// TwinCAT 3 PLC project CarlPlc
// ProgramVersion: 3.1.4022.1
// libraries:
//   Tc2_ModbusRTU, * (Beckhoff Automation GmbH)
//   Tc2_Standard, * (Beckhoff Automation GmbH)
//   Tc2_System, * (Beckhoff Automation GmbH)
//   Tc2_Utilities, * (Beckhoff Automation GmbH)
//   Tc3_Module, * (Beckhoff Automation GmbH)
//   BASIC,3.3.3.0,OSCAT
// project tree:
//   Common/ DetectEvent.TcPOU (not stored), GVL_Common.TcGVL, TasterEventStates.TcDUT (not stored), TasterEventType.TcDUT (not stored), LinearCalibration.TcDUT (not stored)
//   FlowRateSensor/ GVL_FlowControl.TcGVL (not stored), PRG_UpdateFlowRateSensor.TcPOU (not stored)
//   GasAnalysis/ GVL_GasAnalysis.TcGVL (not stored), PRG_GasAnalysis.TcPOU
//   GasSupply/ GVL_GasSupply.TcGVL (not stored), PRG_UpdateGasSupply.TcPOU
//   MotorControl/ GVL_MotorControl.TcGVL (not stored), PRG_UpdateMotor.TcPOU (not stored)
//   pHOrpControl/ EN_ModbusReadTarget.TcDUT (not stored), GVL_PhOrpControl.TcGVL (not stored), PRG_ReadModbusSensorData.TcPOU (not stored), PRG_UpdatePhControl.TcPOU (not stored)
//   / PlcTask.TcTTO
//   MAIN/ MAIN.TcPOU
//   ReactorPressureControl/ GVL_ReactorPressureControl.TcGVL, PRG_UpdatePressureSensor.TcPOU
//   RoomTempRh/ GVL_TempRHSensor.TcGVL (not stored), PRG_UpdateRoomTempRh.TcPOU (not stored)
//   Systemidentifikation/ Messung1.TcPOU, Messung2.TcPOU
//   TemperatureControl/ EN_TempControlMode.TcDUT (not stored), GVL_TemperatureControl.TcGVL, FUN_ComputeMovingSetPoint.TcPOU (not stored), PRG_UpdateTemperatureControl.TcPOU
//   TemperatureControl/PID/ CLK_PRG.TcPOU (not stored), FB_PWM.TcPOU, FT_DERIV.TcPOU (not stored), FT_PIDWL.TcPOU (not stored), FT_PIWL.TcPOU (not stored), PWM_DC.TcPOU (not stored), TP_X.TcPOU, T_PLC_MS.TcPOU, T_PLC_US.TcPOU (not stored)
// real-time tasks:
//   TASK PlcTask: cycle T#10ms, priority 20, ADS port 350
// I/O:
//   DEVICE Device 1 (EtherCAT), AmsNetId 5.54.16.198.2.1
//     Term 1 (EK1200) [EK1200-5000 EtherCAT Power supply (2A E-Bus)]
//       Term 2 (EL3014) Motor Speed In [EL3014 4Ch. Ana. Input 0-20mA DIFF]
//       Term 3 (EL4004) Motor Speed Out [EL4004 4Ch. Ana. Output 0-10V, 12bit]
//       Term 4 (EL2004) DO Heating Cooling [EL2004 4Ch. Dig. Output 24V, 0.5A]
//       Term 5 (EL2004) DO Gassing Valves [EL2004 4Ch. Dig. Output 24V, 0.5A]
//       Term 6 (EL2004) DO Motor Control Out [EL2004 4Ch. Dig. Output 24V, 0.5A]
//       Term 7 (EL6021) PhModbus [EL6021 Interface (RS422/485)]
//       Term 8 (EL6021) OrpModbus [EL6021 Interface (RS422/485)]
//       Term 21 (EL1004) DI Gas Analysis [EL1004 4Ch. Dig. Input 24V, 3ms]
//       Term 18 (EL3052) AI Pressure Flow [EL3052 2Ch. Ana. Input 4-20mA]
//       Term 24 (EL3052) AI Heating Cooling [EL3052 2Ch. Ana. Input 4-20mA]
//       Term 10 (EL9184) [EL9184 Potential Connection, 8 x 24V, 8 x Ground]
//       Term 26 (EL3044) [EL3044 4Ch. Ana. Input 0-20mA]
//       Term 9 (EL9011) [EL9011 End Terminal]
// variable links:
//   CarlPlc/CarlPlc Instance <-> Device 1 (EtherCAT)/Term 1 (EK1200)/Term 18 (EL3052) AI Pressure Flow
//     PlcTask Inputs/GVL_FlowControl.flowRateRawCounts <-> FlowRateSensor/FlowRateRaw
//     PlcTask Inputs/GVL_ReactorPressureControl.pressureRawCounts <-> PressureSensor/PressureSensorRaw
//   CarlPlc/CarlPlc Instance <-> Device 1 (EtherCAT)/Term 1 (EK1200)/Term 2 (EL3014) Motor Speed In
//     PlcTask Inputs/GVL_MotorControl.motorActualSpeed <-> AI Motor RPM/Value
//     PlcTask Inputs/GVL_TempRHSensor.roomRhRaw <-> AI Room RH/Value
//     PlcTask Inputs/GVL_TempRHSensor.roomTempRaw <-> AI Room Temp/Value
//   CarlPlc/CarlPlc Instance <-> Device 1 (EtherCAT)/Term 1 (EK1200)/Term 21 (EL1004) DI Gas Analysis
//     PlcTask Inputs/GVL_GasAnalysis.ch4FlowSensor <-> Flow Sensor CH4/Input
//     PlcTask Inputs/GVL_GasAnalysis.o2FlowSensor <-> Flow Sensor O2/Input
//   CarlPlc/CarlPlc Instance <-> Device 1 (EtherCAT)/Term 1 (EK1200)/Term 24 (EL3052) AI Heating Cooling
//     PlcTask Inputs/GVL_TemperatureControl.jacketTempRaw <-> AI Jacket Temp/Value
//   CarlPlc/CarlPlc Instance <-> Device 1 (EtherCAT)/Term 1 (EK1200)/Term 26 (EL3044)
//     PlcTask Inputs/GVL_GasAnalysis.ch4SensorRaw <-> AI CH4/Value
//     PlcTask Inputs/GVL_GasAnalysis.o2SensorRaw <-> AI O2/Value
//     PlcTask Inputs/GVL_GasSupply.gasSupplyPressureRaw <-> AI Gas Supply Pressure/Value
//   CarlPlc/CarlPlc Instance <-> Device 1 (EtherCAT)/Term 1 (EK1200)/Term 3 (EL4004) Motor Speed Out
//     PlcTask Outputs/GVL_MotorControl.motorTargetSpeed <-> MotorTargetSpeed/MotorTargetSpeed
//     PlcTask Outputs/GVL_PhOrpControl.acidPumpSpeedCount <-> AcidPumpSpeedCount/acidPumpSpeedCount
//   CarlPlc/CarlPlc Instance <-> Device 1 (EtherCAT)/Term 1 (EK1200)/Term 4 (EL2004) DO Heating Cooling
//     PlcTask Outputs/GVL_TemperatureControl.coldValve <-> ColdValve/Output
//     PlcTask Outputs/GVL_TemperatureControl.hotValve <-> HotValve/Output
//     PlcTask Outputs/GVL_TemperatureControl.pumpOn <-> PumpOn/Output
//     PlcTask Outputs/GVL_TemperatureControl.steriValve <-> SteriValve/Output
//   CarlPlc/CarlPlc Instance <-> Device 1 (EtherCAT)/Term 1 (EK1200)/Term 5 (EL2004) DO Gassing Valves
//     PlcTask Outputs/GVL_GasSupply.gasSupplyValve <-> GasSupplyValve/Output
//     PlcTask Outputs/GVL_ReactorPressureControl.reactorPressureInletValve <-> reactorPressureInlet/ReactorPressureInlet
//     PlcTask Outputs/GVL_ReactorPressureControl.reactorPressureOutletValve <-> reactorPressureOutlet/Output
//   CarlPlc/CarlPlc Instance <-> Device 1 (EtherCAT)/Term 1 (EK1200)/Term 6 (EL2004) DO Motor Control Out
//     PlcTask Outputs/GVL_MotorControl.motorReset <-> motorReset/Output
//     PlcTask Outputs/GVL_MotorControl.motorStart <-> motorStart/Output
//   CarlPlc/CarlPlc Instance <-> Device 1 (EtherCAT)/Term 1 (EK1200)/Term 7 (EL6021) PhModbus
//     PlcTask Inputs/GVL_Common.PhModbus.InData/D[{0..21}] <-> COM TxPDO-Map Inputs/Data In {0..21}  (22 links)
//     PlcTask Inputs/GVL_Common.PhModbus.InData/Status <-> COM TxPDO-Map Inputs/Status
//     PlcTask Outputs/GVL_Common.PhModbus.OutData/Ctrl <-> COM RxPDO-Map Outputs/Ctrl
//     PlcTask Outputs/GVL_Common.PhModbus.OutData/D[{0..21}] <-> COM RxPDO-Map Outputs/Data Out {0..21}  (22 links)
//   CarlPlc/CarlPlc Instance <-> Device 1 (EtherCAT)/Term 1 (EK1200)/Term 8 (EL6021) OrpModbus
//     PlcTask Inputs/GVL_Common.OrpModbus.InData/D[{0..21}] <-> COM TxPDO-Map Inputs/Data In {0..21}  (22 links)
//     PlcTask Inputs/GVL_Common.OrpModbus.InData/Status <-> COM TxPDO-Map Inputs/Status
//     PlcTask Outputs/GVL_Common.OrpModbus.OutData/Ctrl <-> COM RxPDO-Map Outputs/Ctrl
//     PlcTask Outputs/GVL_Common.OrpModbus.OutData/D[{0..21}] <-> COM RxPDO-Map Outputs/Data Out {0..21}  (22 links)

CONFIGURATION CarlPlc
    RESOURCE PLC ON TwinCAT3
        TASK PlcTask(INTERVAL := T#10ms, PRIORITY := 20);
        PROGRAM MAIN WITH PlcTask : MAIN;
    END_RESOURCE
END_CONFIGURATION

// ---- Common/GVL_Common.TcGVL
VAR_GLOBAL
	
	loopCounter					: INT := 0;
	
		
	(* pH, ORP, and integrated thermometers *)
	PhModbus					: ModbusRtuMaster_KL6x22B;
	OrpModbus 					: ModbusRtuMaster_KL6x22B;
	PhValueArrayIn				: ARRAY [0..9]OF REAL;
	TPhValueArrayIn				: ARRAY [0..9]OF REAL;
	OrpValueArrayIn				: ARRAY [0..9] OF REAL;
	TOrpValueArrayIn			: ARRAY [0..9] OF REAL;
	
	
	
	
	
	
	
	
END_VAR

// ---- ReactorPressureControl/GVL_ReactorPressureControl.TcGVL
VAR_GLOBAL
	
	(* gas in-flow valve *)	
	reactorPressureInletValve AT %Q*	: BOOL := FALSE;
	
	(* gas out-flow bypass valve *)
	reactorPressureOutletValve		AT %Q* 	: BOOL := FALSE;

	(* pressure sensor *)
	pressureRawCounts	AT %I*	: INT := 0;
	pressureSensorCalibration	: LinearCalibration := (scaleFactor := 2.1626297577854671280276816608997E-4, offset := -1.0);
	pressureBar					: REAL := 0.0;
	pressureStart				: BOOL := FALSE;
	pressureStop				: BOOL := FALSE;

END_VAR

VAR_GLOBAL PERSISTENT
	pressureSetBar				: REAL;
	pressureRunning				: BOOL := FALSE;
END_VAR

// ---- TemperatureControl/GVL_TemperatureControl.TcGVL
VAR_GLOBAL

	tPhCurrent					: REAL := 0.0;
	tPhLastReadingValid			: BOOL := FALSE;
	tOrpCurrent					: REAL := 0.0;
	tOrpLastReadingValid		: BOOL := FALSE;


	(* temperature control *)
	pumpOn				AT %Q* 	: BOOL := FALSE;
	coldValve			AT %Q* 	: BOOL := FALSE;
	hotValve			AT %Q* 	: BOOL := FALSE;
	steriValve			AT %Q*	: BOOL := FALSE; 
	
	jacketTempRaw		AT %I*	: INT;
	jacketTempC					: REAL := 0.0;
	jacketTempK					: REAL := 0.0;
	
	
	tempControlStop				: BOOL := FALSE;
	tempControlStart			: BOOL := FALSE;
	hotValveButton				: BOOL := FALSE;
	coldValveButton				: BOOL := FALSE;
	
	pumpIsRunning				: BOOL := FALSE;
	tempControlRunning			: BOOL := FALSE;
	tempSafetyEnabled			: BOOL := FALSE;
	
	steriStart					: BOOL := FALSE;
	steriStop					: BOOL := FALSE;
	steriRunning				: BOOL := FALSE;

	
	currentMeanTemp				: REAL := 0;
	currentTempValid			: BOOL := FALSE;
	(* target temp -> see retains *) 
	
	tempIsBelowSteriTemp		: BOOL := TRUE;
	(* target steri temp --> see retains *)	

	
END_VAR

VAR_GLOBAL PERSISTENT
	targetControlTemp			: REAL;
	targetSteriTemp				: REAL;
	targetSteriTimeMinutes		: INT;
	remainingSteriTimeMinutes	: REAL;
	
	
	remainingSteriTimeInMs		: DINT; (* 30 min in ms *)
	
	countTempSpikes				: INT;
	countValveMaxTimeExceeded	: INT;

	pidResetCounter				: INT;
END_VAR

// ---- MAIN/MAIN.TcPOU
PROGRAM MAIN
VAR


END_VAR

loopCounter := loopCounter + 1;

PRG_ReadModbusSensorData();			//Temperatur von der Ph-Sonde

(* PRG_HandleUserInputs(); *)

PRG_UpdateMotor();					//Rührmotor

//PRG_UpdateTemperatureControl();		

PRG_UpdatePressureSensor();
PRG_UpdateFlowRateSensor();

Messung1();
//Messung2();

//PRG_UpdatePhControl();
//PRG_UpdateGasSupply();			//Erste Messung nicht nötig
//PRG_UpdateRoomTempRh();			//In Messungen implementiert
//PRG_GasAnalysis();				//Nicht notwendig

END_PROGRAM

// ---- ReactorPressureControl/PRG_UpdatePressureSensor.TcPOU
PROGRAM PRG_UpdatePressureSensor
VAR
	evtPressureControlStart		: DetectEvent;
	evtPressureControlStop		: DetectEvent;
	
END_VAR

(* convert the pressure signal *)
pressureBar := INT_TO_REAL(pressureRawCounts)*pressureSensorCalibration.scaleFactor + pressureSensorCalibration.offset;


(* button events *)
evtPressureControlStart(newSignalValue := pressureStart);
evtPressureControlStop(newSignalValue := pressureStop);

IF evtPressureControlStart.eventDetected = TASTEVT_PositiveEdge THEN
	pressureStart := FALSE;
	pressureRunning := TRUE;
END_IF

IF evtPressureControlStop.eventDetected = TASTEVT_PositiveEdge THEN
	pressureStop := FALSE;
	pressureRunning := FALSE;
END_IF


(* controller *)
IF pressureRunning THEN
	IF pressureBar > pressureSetBar + 0.01  THEN
		reactorPressureInletValve := FALSE;
	END_IF
	
	IF pressureBar < pressureSetBar - 0.01 THEN
		reactorPressureInletValve := TRUE;
	END_IF
ELSE
	reactorPressureInletValve := FALSE;
END_IF

END_PROGRAM

// ---- Systemidentifikation/Messung1.TcPOU
PROGRAM Messung1
VAR
	//PWM Settings
	pwmPeriodinSec			: TIME 	:= T#25S;
	pwmDutyCycle			: REAL 	:= 0.0;	
	pwmOutputValveControl 	: FB_PWM;
	status 					: INT 	:= 0; 			//Status 0 : Initial 
													//Status 1 : Heating to Startpoint
													//Status 2 : Heating while recording
													//Status 3 : Cooling while recording
													//STatus is set manuelly
													
END_VAR


(*Temperature should be increased to a value in a first step. 
This is to serve as a 0 point. In the second step, the duty cycle is increased and the step response is recorded.  
The container is then closed. The same duty cycle is used.
Finally, the water is cooled with a DutyCycle of ... .
*)

(* jacket temperature input *)
jacketTempC := INT_TO_REAL(jacketTempRaw)/32768.0*200.0 -50.0;
(* room temperature input *) //Is not in use in TemperaturControl
roomTemp := (INT_TO_REAL(roomTempRaw)/32767.0)*100.0 - 40.0;  (* Sensor Range: -40°C to + 60°C *)



// DutyCycle - To get a startingTemp.
CASE status OF
	
	//------Initial - Status 0----------//
	0:
	(* Setting Valves & Pump off  *)
	pumpOn := FALSE;
	coldValve := FALSE;
	hotValve := FALSE;
	steriValve := FALSE;
	
	//------HEATING - Status 1----------//
	1:
	//Starting pump
	pumpOn := TRUE;
	
	//DutyCyle for startpoint
	pwmDutyCycle:= 20 ;
	pwmOutputValveControl(pwmCycleTime:=pwmPeriodinSec, pwmDutyCycle:=pwmDutyCycle); //Gets the Output
	hotValve := pwmOutputValveControl.Q;
	
	
	//------HEATING - Status 2----------//
	2:	
	//DutyCycle for step response
	pwmDutyCycle:= 40 ;
	pwmOutputValveControl(pwmCycleTime:=pwmPeriodinSec, pwmDutyCycle:=pwmDutyCycle); //Gets the Output
	hotValve := pwmOutputValveControl.Q;
	
	//------COOLING - Status 3----------//
	3:
	//Turning off hotValve
	hotValve := FALSE;
	
	//DutyCycle for cooling
	pwmDutyCycle:= 40 ;
	pwmOutputValveControl(pwmCycleTime:=pwmPeriodinSec, pwmDutyCycle:=pwmDutyCycle); //Gets the Output
	coldValve := pwmOutputValveControl.Q;
END_CASE

END_PROGRAM

// ---- TemperatureControl/PID/FB_PWM.TcPOU
FUNCTION_BLOCK FB_PWM
VAR_INPUT
	pwmCycleTime 		: TIME := T#10S;
	pwmDutyCycle		: REAL := 0.5;
	reset				: BOOL := FALSE;
END_VAR
VAR_OUTPUT
	Q					: BOOL := FALSE;
END_VAR
VAR
	pwmTimeInMs			: INT	:= 0;
	pwmTimer		: TON;
	pwmLowTimer			: TON;
	dutyCycleInMs		: TIME;
	test				: INT;
	internalReset 		: BOOL := FALSE;
END_VAR

IF pwmDutyCycle < 0 THEN
	pwmDutyCycle := 0.0;
END_IF

IF reset OR internalReset THEN
	pwmTimer(IN:= FALSE);
	reset := FALSE;
	internalReset := FALSE;
ELSE
	pwmTimeInMs := TIME_TO_INT(pwmCycleTime);
	IF Q THEN
		(* high  --> running falling timer *)
		dutyCycleInMs := INT_TO_TIME(REAL_TO_INT(INT_TO_REAL(pwmTimeInMs)*pwmDutyCycle));
		pwmTimer(IN:=TRUE, PT:=dutyCycleInMs);
		IF pwmTimer.Q THEN
			internalReset := TRUE;
			Q := FALSE;
		END_IF		
	ELSE
		(* low --> running rising timer *)
		dutyCycleInMs := INT_TO_TIME(REAL_TO_INT(INT_TO_REAL(pwmTimeInMs)*(1.0-pwmDutyCycle)));
		pwmTimer(IN:=TRUE, PT:=dutyCycleInMs);
		IF pwmTimer.Q THEN
			internalReset := TRUE;
			Q := TRUE;
		END_IF		
	END_IF
END_IF

END_FUNCTION_BLOCK

// ---- GasAnalysis/PRG_GasAnalysis.TcPOU
PROGRAM PRG_GasAnalysis
VAR
	evtGasAnalysisStartStop		: DetectEvent;
	evtGasAnalysisManualValve 	: DetectEvent;
END_VAR

ch4ValuemA := ch4SensorRaw*ch4CalibrationToMa.scaleFactor + ch4CalibrationToMa.offset;
ch4ValuePercent := (ch4ValuemA-4.0)*(100.0/16.0);

o2ValuemA := o2SensorRaw*o2CalibrationToMa.scaleFactor + o2CalibrationToMa.offset;
o2ValuePercent := (o2ValuemA-4.0)*(25.0/16.0);



(* CH4 Sensor Status*)
IF ch4ValuemA > 3.9 THEN
	(* running *)
	ch4SensorStatus := 4;
ELSIF (ch4ValuemA < 3.2 AND ch4ValuemA > 2.8) THEN
	(* startup *)
	ch4SensorStatus := 3;
ELSIF (ch4ValuemA < 2.2 AND ch4ValuemA > 1.8) THEN
	(* beam block *)
	ch4SensorStatus := 2;
ELSIF (ch4ValuemA < 1.2 AND ch4ValuemA > 0.8) THEN
	(* fault *)
	ch4SensorStatus := 1;
ELSE
	(* offline *)
	ch4SensorStatus := 0;
END_IF

(* control switches *) 
evtGasAnalysisStartStop(newSignalValue := gasAnalysisControlStartStop);
IF evtGasAnalysisStartStop.eventDetected = TASTEVT_PositiveEdge THEN
	gasAnalysisControlRunning := TRUE;
END_IF

IF evtGasAnalysisStartStop.eventDetected = TASTEVT_NegativeEdge THEN
	gasAnalysisControlRunning := FALSE;
END_IF


IF gasAnalysisControlRunning THEN
	IF ch4ValuePercent > ch4ValuePercentSet  THEN
		gasAnalysisValveAutomatic := TRUE;
	END_IF
	
	IF ch4ValuePercent < ch4ValuePercentSet -1  THEN
		gasAnalysisValveAutomatic := FALSE;
	END_IF
ELSE 
	gasAnalysisValveAutomatic := FALSE;
END_IF


evtGasAnalysisManualValve(newSignalValue := gasAnalysisControlManual);
IF evtGasAnalysisManualValve.eventDetected = TASTEVT_PositiveEdge THEN
	gasAnalysisValveManual := TRUE;
END_IF

IF evtGasAnalysisManualValve.eventDetected = TASTEVT_NegativeEdge THEN
	gasAnalysisValveManual := FALSE;
END_IF

reactorPressureOutletValve := gasAnalysisValveManual OR gasAnalysisValveAutomatic;

END_PROGRAM

// ---- GasSupply/PRG_UpdateGasSupply.TcPOU
PROGRAM PRG_UpdateGasSupply
VAR
	evtGasSupplyStart		: DetectEvent;
	evtGasSupplyStop		: DetectEvent;
END_VAR

gasSupplyPressureBar := INT_TO_REAL(gasSupplyPressureRaw)*gasSupplyPressureSensorCalibration.scaleFactor + gasSupplyPressureSensorCalibration.offset;


(* button events *)
evtGasSupplyStart(newSignalValue := gasSupplyStart);
evtGasSupplyStop(newSignalValue := gasSupplyStop);

IF evtGasSupplyStart.eventDetected = TASTEVT_PositiveEdge THEN
	gasSupplyStart := FALSE;
	gasSupplyRunning := TRUE;
END_IF

IF evtGasSupplyStop.eventDetected = TASTEVT_PositiveEdge THEN
	gasSupplyStop := FALSE;
	gasSupplyRunning := FALSE;
END_IF


IF gasSupplyRunning THEN
	IF gasSupplyPressureBar > gasSupplyPressureSetBar + 0.1 THEN
		gasSupplyValve := FALSE;
	END_IF
	
	IF gasSupplyPressureBar < gasSupplyPressureSetBar - 0.1 THEN
		gasSupplyValve := TRUE;
	END_IF
 
END_IF

END_PROGRAM

// ---- Systemidentifikation/Messung2.TcPOU
PROGRAM Messung2
VAR
	//PWM Settings
	pwmPeriodinSec			: TIME 	:= T#25S;
	pwmDutyCycle			: REAL 	:= 0.0;	
	pwmOutputValveControl 	: FB_PWM;
	status 					: INT 	:= 0; 			//Status 0 : Initial 
													//Status 1 : Heating to Startpoint
													//Status 2 : Heating while recording
													//Status 3 : Cooling while recording
													//STatus is set manuelly
													
END_VAR


(*Temperature should be increased to a value in a first step. 
This is to serve as a 0 point. should be around 70°C
In the second step, the duty cycle is increased and the step response is recorded while the container is closed.
Finally, the water is cooled with a DutyCycle of ... .
*)

(* jacket temperature input *)
jacketTempC := INT_TO_REAL(jacketTempRaw)/32768.0*200.0 -50.0;
(* room temperature input *) //Is not in use in TemperaturControl
roomTemp := (INT_TO_REAL(roomTempRaw)/32767.0)*100.0 - 40.0;  (* Sensor Range: -40°C to + 60°C *)


// DutyCycle - To get a startingTemp.
CASE status OF
	
	//------Initial - Status 0----------//
	0:
	(* Setting Valves & Pump off  *)
	pumpOn := FALSE;
	coldValve := FALSE;
	hotValve := FALSE;
	steriValve := FALSE;
	
	//------HEATING - Status 1----------//
	1:
	//Starting pump
	pumpOn := TRUE;
	
	//DutyCyle for startpoint
	pwmDutyCycle:= 40 ;
	pwmOutputValveControl(pwmCycleTime:=pwmPeriodinSec, pwmDutyCycle:=pwmDutyCycle); //Gets the Output
	hotValve := pwmOutputValveControl.Q;
	
	
	//------HEATING - Status 2----------//
	2:	
	//Turning off the pump
	pumpOn := FALSE;
	
	//DutyCycle for step response
	pwmDutyCycle:= 80 ;
	pwmOutputValveControl(pwmCycleTime:=pwmPeriodinSec, pwmDutyCycle:=pwmDutyCycle); //Gets the Output
	steriValve := pwmOutputValveControl.Q;
	
	//------COOLING - Status 3----------//
	3:
	//Turning off hotValve & steriValve
	hotValve := FALSE;
	steriValve := FALSE;
	
	//DutyCycle for cooling
	pwmDutyCycle:= 40 ;
	pwmOutputValveControl(pwmCycleTime:=pwmPeriodinSec, pwmDutyCycle:=pwmDutyCycle); //Gets the Output
	coldValve := pwmOutputValveControl.Q;
END_CASE

END_PROGRAM

// ---- TemperatureControl/PID/TP_X.TcPOU
FUNCTION_BLOCK TP_X
VAR_INPUT
	IN : BOOL;
	PT : TIME;
END_VAR
VAR_OUTPUT
	Q : BOOL;
	ET : TIME;
END_VAR
VAR
	edge : BOOL;
	start : TIME;
	tx: TIME;
END_VAR

(*retriggerable edge triggered pulse similar to TP but with a retrigger function
if the pt input is 0 then output is always low.
*)

(* read system_time *)
tx := DWORD_TO_TIME(T_PLC_MS());

(* rising edge trigger *)
IF IN AND NOT edge THEN
	start := tx;
	Q := PT > t#0ms;
ELSIF Q THEN
	ET := tx - start;
	IF ET >= PT THEN
		Q := FALSE;
		ET := t#0ms;
	END_IF;
END_IF;
edge := IN;

END_FUNCTION_BLOCK

// ---- TemperatureControl/PID/T_PLC_MS.TcPOU
FUNCTION T_PLC_MS : DWORD
VAR CONSTANT
	debug : BOOL := 0;
	N : INT := 0;
	offset : DWORD := 0;
END_VAR
VAR
	tx : TIME;
END_VAR

(*T_PLC_MS reads the internal PLC timer and return the time, it has the advantage to be able to set a debug mode 
and speed up the counter to test the plc timer overrun which occurs every 50 days respectively 25 days at siemens S7
this routine also allows to correct the behavior of s7 where the internal plc counter will not count all 32 bits.

*)

tx := TIME();
T_PLC_MS := TIME_TO_DWORD(Tx);

IF debug THEN
	T_PLC_MS := (SHL(T_PLC_MS,N) OR SHL(DWORD#1,N)-1) + OFFSET;
END_IF;

END_FUNCTION

// ---- TemperatureControl/PRG_UpdateTemperatureControl.TcPOU
PROGRAM PRG_UpdateTemperatureControl
VAR
	tempControlMode				: EN_TempControlMode := EN_TempControlMode.TEMP_MODE_MANUAL;  

	(* Controller settings *)
	pwmPeriodinSec			: TIME := T#25S;
	pwmDutyCycle			: REAL := 0.0;	
	pwmOutputValveControl 	: FB_PWM;
	
	pidController			: FT_PIDWL;
	
	kp_heating				: REAL := 0.002;
	tv_heating				: REAL := 200;
	tn_heating				: REAL := 1800;
	
	kp_cooling				: REAL := 0.006;
	tv_cooling				: REAL := 200;
	tn_cooling				: REAL := 1800;

	kp_steri				: REAL := 0.0065;
	tv_steri				: REAL := 200;
	tn_steri				: REAL := 300;
	
	kp						: REAL := kp_heating;
	tv						: REAL := tv_heating;
	tn						: REAL := tn_heating;

	(* KD = KP*TV *)			
	(* KI = KP/TN *)
	
	errorTemp				: REAL := 0.0;
	pidReset				: BOOL := FALSE;
		
	evtSteriStart			: DetectEvent;
	evtSteriStop			: DetectEvent;
		
	evtTempControlStart		: DetectEvent;
	evtTempControlStop		: DetectEvent;
	
	windUpResetTimer		: TON;
	windUpResetTime			: TIME := T#30S;
	
	maxValveOnTimer		 	: TON;
	maxValveOnTime			: TIME := T#25S;	
	
	evtPidReset				: DetectEvent;
	(*
	myPwmBlock				: FB_PWM;
	pwmCycleTime			: TIME := T#2S;
	myPwmDutyCycle			: REAL := 0.5;
	*)
END_VAR

(* jacket temperature input *)
jacketTempC := INT_TO_REAL(jacketTempRaw)/32768.0*200.0 -50.0;



evtSteriStart(		newSignalValue := steriStart);
evtSteriStop(		newSignalValue := steriStop);
evtTempControlStart(newSignalValue := tempControlStart);
evtTempControlStop(	newSignalValue := tempControlStop);
evtPidReset( 		newSignalValue := pidReset);


IF evtSteriStart.eventDetected = TASTEVT_PositiveEdge THEN
	steriStart := FALSE;
	pumpOn := FALSE;
	pidController( RST:= TRUE );
	tempControlMode	:= EN_TempControlMode.TEMP_MODE_STERI;
	tempControlRunning := FALSE;
	steriRunning := TRUE;
	steriValve := FALSE;
	coldValve := FALSE;
	hotValve := FALSE;
	(* Set remaining steri temp *)
	remainingSteriTimeInMs := targetSteriTimeMinutes*60*1000; 
END_IF

IF evtTempControlStart.eventDetected = TASTEVT_PositiveEdge THEN
	tempControlStart := FALSE;
	pumpOn := FALSE;
	pidController( RST:= TRUE );
	tempControlMode	:= EN_TempControlMode.TEMP_MODE_HEATCOOL;
	tempControlRunning := TRUE;
	steriRunning := FALSE;
	steriValve := FALSE;
	coldValve := FALSE;
	hotValve := FALSE;
END_IF

IF 	evtSteriStop.eventDetected = TASTEVT_PositiveEdge OR
 	evtTempControlStop.eventDetected = TASTEVT_PositiveEdge 
THEN
	steriStop := FALSE;
	tempControlStop := FALSE;
	pumpOn := FALSE;
	pidController( RST:= TRUE );
	tempControlRunning := FALSE;
	steriRunning := FALSE;
	tempControlMode	:= EN_TempControlMode.TEMP_MODE_MANUAL;
	coldValve := FALSE;
	hotValve := FALSE;
	steriValve := FALSE;
	(* TODO: Reset Steri Timer *)
END_IF

CASE tempControlMode OF
	EN_TempControlMode.TEMP_MODE_MANUAL:
		pumpOn := FALSE;
		pidController( RST:= TRUE );
		
	EN_TempControlMode.TEMP_MODE_HEATCOOL:
	
		
		pumpOn := TRUE;
		(* errorTemp := targetControlTemp - currentMeanTemp; *)
		errorTemp := FUN_ComputeMovingSetPoint(currentTemp := currentMeanTemp, targetSetPoint := targetControlTemp) - currentMeanTemp;
		
		pidController(	IN:= errorTemp,
						KP:= kp,
						TN:= tn,
						TV:= tv,
						LIM_L:= -1.0,
						LIM_H:= 1.0,
						RST:= pidReset);
						
		pwmDutyCycle := ABS(pidController.Y); (* !! pwm block cannot handle negative inputs *)
		pwmOutputValveControl(pwmCycleTime:=pwmPeriodinSec, pwmDutyCycle:=pwmDutyCycle);
		
		IF pidController.Y > 0 THEN
			(* heating *)
			coldValve := FALSE;
			hotValve := pwmOutputValveControl.Q;
			kp := kp_heating;
			tv := tv_heating;
			tn := tn_heating;
			
		ELSE
			(* cooling *)
			coldValve := pwmOutputValveControl.Q;
			hotValve := FALSE;

			kp := kp_cooling;
			tv := tv_cooling;
			tn := tn_cooling;
		END_IF
		
	
	EN_TempControlMode.TEMP_MODE_STERI:
		pumpOn := FALSE;
		errorTemp := targetSteriTemp - currentMeanTemp;
		pidController(	IN:= errorTemp,
						KP:= kp_steri,
						TN:= tn_steri,
						TV:= tv_steri,
						LIM_L:= -1.0,
						LIM_H:= 1.0,
						RST:= pidReset);
						
		pwmDutyCycle := ABS(pidController.Y); (* !! pwm block cannot handle negative inputs *)
		
		pwmOutputValveControl(pwmCycleTime:=pwmPeriodinSec, pwmDutyCycle:=pwmDutyCycle);
				
		IF pidController.Y > 0 THEN
			(* heating *)
			coldValve := FALSE;
			steriValve := pwmOutputValveControl.Q;
		ELSE
			(* cooling *)
			(* coldValve := pwmOutputValveControl.Q; *)
			steriValve := FALSE;
		END_IF
		
		IF currentMeanTemp > (targetSteriTemp-0.5) THEN
			(* count down 10 ms each cycle *)
			remainingSteriTimeInMs := remainingSteriTimeInMs - 10;
			IF remainingSteriTimeInMs < 0 THEN
				tempControlMode := EN_TempControlMode.TEMP_MODE_MANUAL;
				steriValve := FALSE;
				coldValve := FALSE;
				steriStop := TRUE;
			END_IF
		END_IF		
		remainingSteriTimeMinutes := DINT_TO_REAL(remainingSteriTimeInMs)/(60.0*1000.0);
	
	
END_CASE

(*
maxValveOnTimer(IN:= (coldValve OR hotValve OR steriValve), PT:= maxValveOnTime);
IF maxValveOnTimer.Q THEN
	maxValveOnTimer(IN:=FALSE);
	countValveMaxTimeExceeded := countValveMaxTimeExceeded + 1;
	pidReset := TRUE;
	steriValve := FALSE;
	coldValve := FALSE;
	hotValve := FALSE;
END_IF
*)
(*
IF tempSafetyEnabled THEN
	IF (tPhLastReadingValid = FALSE AND tOrpLastReadingValid = FALSE) OR
		(currentMeanTemp > targetControlTemp + 0.5 OR currentMeanTemp < targetControlTemp - 0.5) THEN
		//tempControlMode := EN_TempControlMode.TEMP_MODE_MANUAL;
		pidReset := TRUE;
		countTempSpikes := countTempSpikes + 1;
		steriValve := FALSE;
		coldValve := FALSE;
		hotValve := FALSE;
	END_IF
END_IF
*)
 
IF evtPidReset.eventDetected = TASTEVT_PositiveEdge THEN
	pidReset := FALSE;
	pidController(RST:=TRUE);
	pidResetCounter := pidResetCounter + 1;
	steriValve := FALSE;
	coldValve := FALSE;
	hotValve := FALSE;
END_IF

END_PROGRAM
